(* CoDeSys 2.3.10.0 project: demo.pro *)
(* Libraries: STANDARD.LIB 5.6.98 12:03:02 *)

(* Task configuration *)
TASK Standard (PRIORITY := 0, INTERVAL := T#10ms);
	MAIN
END_TASK

(* Global variable list: Globale_Variablen *)
VAR_GLOBAL
	In_BOOL1 AT%MX0.0 : BOOL;
	In_BOOL2: BOOL;

	In_SINT1: SINT;
	In_SINT2: SINT;
	In_SINT3: SINT;
	In_SINT4: SINT;
	In_INT1: INT;
	In_INT2: INT;
	In_DINT: DINT;
	In_STRING: STRING(11);
	In_TIME: TIME;
	In_REAL: REAL;

	TOD_Test : TOD;
	DT_Test: DT;
	DATE_Test: DATE;

	ArrayOfString: ARRAY[1..5] OF STRING(10);
	ArrayOfBool:  ARRAY[1..5] OF BOOL;

	ArrayOfTestStruct2: ARRAY[1..4] OF ST_Test2;

	TestStruct:  ST_Test;

	ArrayTestStruct3: ARRAY [1..20] OF ST_Test3;

	TestStruct4 :  ST_Test4;

	ArrayChart: ARRAY [1..10] OF ST_ChartFields (*Kommentar*);
END_VAR

(* Data type *)
TYPE ST_ChartFields :
STRUCT
	graph1: INT;
	graph2: INT;
END_STRUCT
END_TYPE

(* Data type *)
TYPE ST_Test :
STRUCT
	nByte: BYTE;
	fReal: REAL;
	iSint: SINT;
	tTime: TIME;
	arrString: ARRAY[1..5] OF STRING(6);
	iInt: INT;
END_STRUCT
END_TYPE

(* Data type *)
TYPE ST_Test2 :
STRUCT
	sString: STRING(5) := 'xxxxx';
	fReal: REAL;
	iSint: SINT;
	iInt: INT;
	arrByte: ARRAY[1..5] OF BYTE;
END_STRUCT
END_TYPE

(* Data type *)
TYPE ST_Test3 :
STRUCT
	sString: STRING(10) := '';
	fReal: REAL;
	iInt: INT;
	nByte: BYTE;
	bCheckbox: BOOL;
	arrBool: ARRAY[1..5] OF BOOL;
END_STRUCT
END_TYPE

(* Data type *)
TYPE ST_Test4 :
STRUCT
	fReal: REAL;
	tTime: TIME;
	tTod: TOD;
	dtDate: DATE;
	arrString: ARRAY[1..5] OF STRING(6);
END_STRUCT
END_TYPE

(* POU MAIN, FBD *)
PROGRAM MAIN
VAR
	fbRamp1: FB_Ramp;
	fbRamp2: FB_Ramp;
	fbShiftArray: FB_ShiftArray;
	fbRunningLight: FB_RunningLight;
	Ramp1 : INT;
	Ramp2 : INT;
	RunningLight1: BOOL;
	RunningLight2: BOOL;
	RunningLight3: BOOL;
	RunningLight4: BOOL;
	RunningLight5: BOOL;
END_VAR
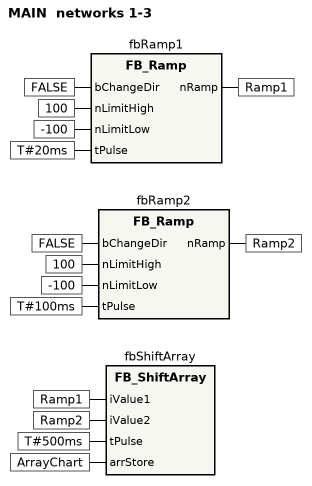
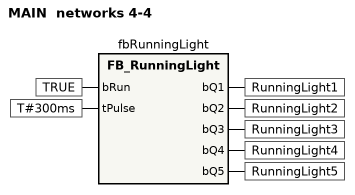
_FBD_ (* Function Block Diagram *)
NETWORK 1
	fbRamp1:FB_Ramp(bChangeDir: FALSE, nLimitHigh: 100, nLimitLow: -100, tPulse: T#20ms) => Ramp1
NETWORK 2
	fbRamp2:FB_Ramp(bChangeDir: FALSE, nLimitHigh: 100, nLimitLow: -100, tPulse: T#100ms) => Ramp2
NETWORK 3
	fbShiftArray:FB_ShiftArray(iValue1: Ramp1, iValue2: Ramp2, tPulse: T#500ms, arrStore: ArrayChart)
NETWORK 4
	fbRunningLight:FB_RunningLight(bRun: TRUE, tPulse: T#300ms, bQ2 => RunningLight2, bQ3 => RunningLight3, bQ4 => RunningLight4, bQ5 => RunningLight5) => RunningLight1
_END_FBD_
(* the same logic as Structured Text *)
(* Network 1 *)
fbRamp1(bChangeDir := FALSE, nLimitHigh := 100, nLimitLow := -100, tPulse := T#20ms);
Ramp1 := fbRamp1.nRamp;
(* Network 2 *)
fbRamp2(bChangeDir := FALSE, nLimitHigh := 100, nLimitLow := -100, tPulse := T#100ms);
Ramp2 := fbRamp2.nRamp;
(* Network 3 *)
fbShiftArray(iValue1 := Ramp1, iValue2 := Ramp2, tPulse := T#500ms, arrStore := ArrayChart);
(* Network 4 *)
fbRunningLight(bRun := TRUE, tPulse := T#300ms);
RunningLight2 := fbRunningLight.bQ2;
RunningLight3 := fbRunningLight.bQ3;
RunningLight4 := fbRunningLight.bQ4;
RunningLight5 := fbRunningLight.bQ5;
RunningLight1 := fbRunningLight.bQ1;
END_PROGRAM

(* POU FB's/FB_Ramp, ST *)
FUNCTION_BLOCK FB_Ramp
VAR_INPUT
	bChangeDir: BOOL;		(*change direction*)
	nLimitHigh: INT:= 32767;	(*limit high*)
	nLimitLow: INT:= -32768;	(*limit low*)
	tPulse: TIME:= T#50ms; 	(*pulse pause time for counter*)
END_VAR
VAR_OUTPUT
	nRamp: INT;
END_VAR
VAR
	rtrigChangeDir: R_TRIG;
	tonPulse: TON;
	rsDown: TogRS;
END_VAR
tonPulse(in:=NOT tonPulse.Q, PT:=tPulse);
rsDown(set:=nRamp >= nLimitHigh, reset1:= nRamp <= nLimitLow, clk:=bChangeDir);

IF tonPulse.Q THEN
	IF rsDown.Q1 THEN
		nRamp := nRamp - 1;
	ELSE
		nRamp := nRamp +1;
	END_IF;
END_IF;
END_FUNCTION_BLOCK

(* POU FB's/TogRS, ST *)
FUNCTION_BLOCK TogRS
VAR_INPUT
	CLK : BOOL;
	SET: BOOL;
	RESET1 : BOOL;
END_VAR
VAR_OUTPUT
	Q1 : BOOL;
	edge : BOOL;
END_VAR
IF RESET1 THEN
	Q1 := 0;
ELSIF SET THEN
	Q1:= 1;
ELSIF CLK AND NOT edge THEN
	Q1 := NOT Q1;
END_IF;
edge := clk;
END_FUNCTION_BLOCK

(* POU FB's/FB_ShiftArray, ST *)
FUNCTION_BLOCK FB_ShiftArray
VAR_INPUT
	iValue1: INT;
	iValue2: INT;
	tPulse: TIME:= T#50ms;
END_VAR
VAR_IN_OUT
	arrStore: ARRAY [1..10] OF ST_ChartFields;
END_VAR
VAR
	tonPulse: TON;
	i: BYTE;
END_VAR
tonPulse(in:=NOT tonPulse.Q, PT:=tPulse);

IF tonPulse.Q THEN
	FOR i := 2 TO 10 DO
 		arrStore[i - 1].graph1  :=arrStore[i].graph1;
		arrStore[i - 1].graph2  :=arrStore[i].graph2;
	END_FOR;
	arrStore[10].graph1 := iValue1;
	arrStore[10].graph2 := iValue2;
END_IF;
END_FUNCTION_BLOCK

(* POU FB's/FB_RunningLight, ST *)
FUNCTION_BLOCK FB_RunningLight
VAR_INPUT
	bRun: BOOL;
	tPulse: TIME:= T#500ms;
END_VAR
VAR_OUTPUT
	bQ1: BOOL;
	bQ2: BOOL;
	bQ3: BOOL;
	bQ4: BOOL;
	bQ5: BOOL;
END_VAR
VAR
	tonPulse: TON;
	bActive: BOOL;
	tmp: BOOL;
END_VAR
tonPulse(in:=NOT tonPulse.Q AND bRun, PT:=tPulse);

IF tonPulse.Q THEN
	bQ5:= bQ4;
	bQ4:= bQ3;
	bQ3:= bQ2;
	bQ2:= bQ1;
	bQ1:= tmp;
	tmp := bQ5;
END_IF;

IF NOT bRun THEN
	bQ1 := FALSE;
	bQ2 := FALSE;
	bQ3 := FALSE;
	bQ4 := FALSE;
	bQ5 := FALSE;
END_IF;

IF bRun AND NOT bActive THEN
	bQ1 := TRUE;
END_IF;

bActive := bRun;
END_FUNCTION_BLOCK
